{attribute 'qualified_only'}
{attribute 'strict'}
TYPE E_Msg_Option :
(
	None := 0,
	OneParam := 1,
	TwoParam := 2
)UINT;
END_TYPE

(* stored: Version 1.1.0.1, ProductVersion 3.1.4024.10
   DUT E_Msg_Option: Id {33908b3d-3f31-4b43-8844-0eb647a9d577} *)
